SUBAPPLICATION Uebung_019b (* Umschalten einer Maske *)
  (* Standard: 61499-2; Description: Copyright (c) 2023 Meisterschulen am Ostbahnhof This program and the accompanying materials are made available under the terms of the Eclipse Public License 2.0 which is available at https://www.eclipse.org/legal/epl-2.0/ SPDX-License-Identifier: EPL-2.0 *)
  (* Version 1.0, 2023-10-23, Franz Höpfinger, Meisterschulen am Ostbahnhof *)
  PACKAGE Uebungen;
  IMPORT isobus::UT::io::Softkey::SoftKeyActivationCode::SK_PRESSED;
  IMPORT Uebungen::const::UT::DefaultPool::AlarmMask_A2_medium;
  IMPORT Uebungen::const::UT::DefaultPool::DataMask_M1;
  IMPORT Uebungen::const::UT::DefaultPool::DataMask_M2;
  IMPORT Uebungen::const::UT::DefaultPool::WorkingSet_0;
  IMPORT isobus::UT::Q::const::IDs::ID_NULL;
  IMPORT logiBUS::io::DI::logiBUS_DI::Input_I1;
  IMPORT logiBUS::io::DI::logiBUS_DI::Input_I2;
  IMPORT logiBUS::io::DI::logiBUS_DI::Input_I3;
  IMPORT logiBUS::io::DI::logiBUS_DI_Events::BUTTON_SINGLE_CLICK;
  IMPORT logiBUS::io::DQ::logiBUS_DO::Output_Q1;
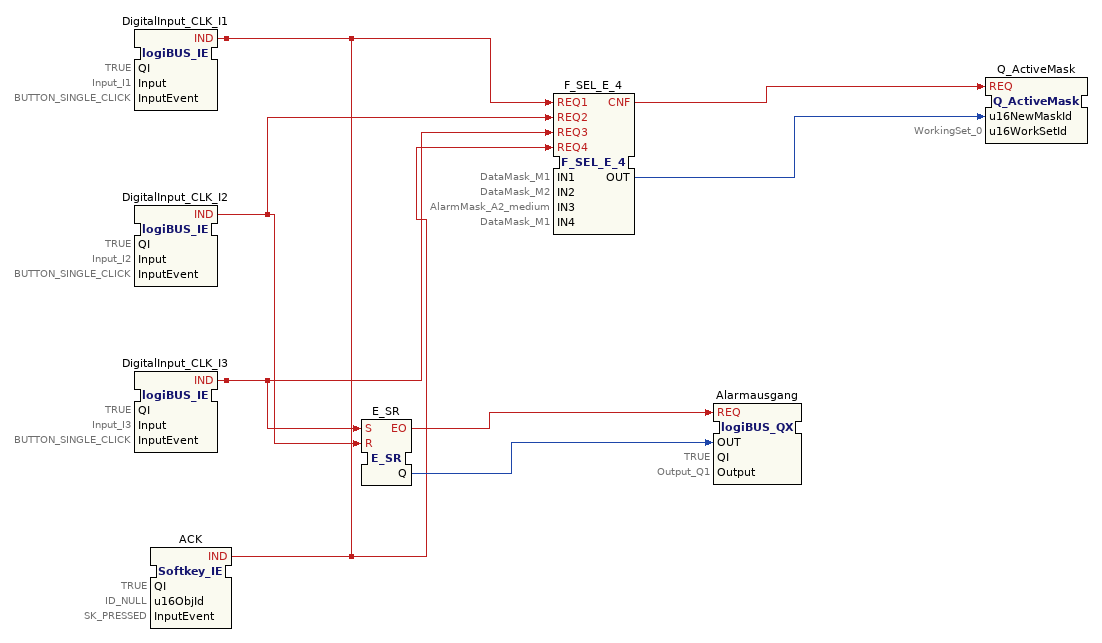
  FBS
    DigitalInput_CLK_I1 : logiBUS::io::DI::logiBUS_IE(QI := TRUE, Input := Input_I1, InputEvent := BUTTON_SINGLE_CLICK);
    Q_ActiveMask : isobus::UT::Q::Q_ActiveMask(u16WorkSetId := WorkingSet_0);
    DigitalInput_CLK_I2 : logiBUS::io::DI::logiBUS_IE(QI := TRUE, Input := Input_I2, InputEvent := BUTTON_SINGLE_CLICK);
    F_SEL_E_4 : eclipse4diac::utils::selection::F_SEL_E_4(IN1 := DataMask_M1, IN2 := DataMask_M2, IN3 := AlarmMask_A2_medium, IN4 := DataMask_M1);
    DigitalInput_CLK_I3 : logiBUS::io::DI::logiBUS_IE(QI := TRUE, Input := Input_I3, InputEvent := BUTTON_SINGLE_CLICK);
    ACK : isobus::UT::io::Softkey::Softkey_IE(QI := TRUE, u16ObjId := ID_NULL, InputEvent := SK_PRESSED);
    E_SR : iec61499::events::E_SR;
    Alarmausgang : logiBUS::io::DQ::logiBUS_QX(QI := TRUE, Output := Output_Q1);
  END_FBS
  EVENT_CONNECTIONS
    DigitalInput_CLK_I1.IND TO F_SEL_E_4.REQ1;
    DigitalInput_CLK_I2.IND TO F_SEL_E_4.REQ2;
    F_SEL_E_4.CNF TO Q_ActiveMask.REQ;
    DigitalInput_CLK_I3.IND TO F_SEL_E_4.REQ3;
    ACK.IND TO F_SEL_E_4.REQ4;
    DigitalInput_CLK_I3.IND TO E_SR.S;
    DigitalInput_CLK_I2.IND TO E_SR.R;
    DigitalInput_CLK_I1.IND TO E_SR.R;
    ACK.IND TO E_SR.R;
    E_SR.EO TO Alarmausgang.REQ;
  END_CONNECTIONS
  DATA_CONNECTIONS
    F_SEL_E_4.OUT TO Q_ActiveMask.u16NewMaskId;
    E_SR.Q TO Alarmausgang.OUT;
  END_CONNECTIONS
END_SUBAPPLICATION
